FUNCTION_BLOCK T_StringSplitterEx
VAR
	SubjectString : TC2_SYSTEM.T_MaxString;
	Delimiter : STRING;
	Delimiter1 : STRING;
	Delimiter2 : STRING;
	NextDelimiterPosition : INT;
	NextDelimiter1Position : INT;
	NextDelimiter2Position : INT;
END_VAR

METHOD GetNext : STRING(255)
VAR_INPUT
END_VAR
VAR
	RemainingLength: INT;
END_VAR
NextDelimiter1Position := FIND(SubjectString , Delimiter1);
NextDelimiter2Position := FIND(SubjectString , Delimiter2);

IF NextDelimiter1Position = 0 THEN
    // use Delimiter 2 position , even if zero...
    NextDelimiterPosition := NextDelimiter2Position;
    Delimiter := Delimiter2;
    
ELSIF NextDelimiter2Position = 0 THEN
    // use Delimiter 1 position , non-zero...
    NextDelimiterPosition := NextDelimiter1Position;
    Delimiter := Delimiter1;

ELSE
    // Both delimters found - use the one nearest the start of the string...
    IF NextDelimiter1Position < NextDelimiter2Position THEN
        NextDelimiterPosition := NextDelimiter1Position;
        Delimiter := Delimiter1;
    ELSE
        NextDelimiterPosition := NextDelimiter2Position;
        Delimiter := Delimiter2;
	END_IF
END_IF

IF NextDelimiterPosition > 0 THEN // delimitter found
    
    // extract next sub-string
	GetNext := LEFT(SubjectString,NextDelimiterPosition - 1);
    
    // remove sub-string from subject string
	RemainingLength := LEN(SubjectString) - NextDelimiterPosition - LEN(Delimiter) + 1;
	SubjectString := RIGHT(SubjectString,RemainingLength);
    
    // strip any delimitters from front of remaining string
    WHILE FIND(SubjectString,Delimiter1) = 1 DO
        SubjectString := RIGHT(SubjectString,LEN(SubjectString) - LEN(Delimiter1));
	END_WHILE
    WHILE FIND(SubjectString,Delimiter2) = 1 DO
        SubjectString := RIGHT(SubjectString,LEN(SubjectString) - LEN(Delimiter2));
	END_WHILE
	
ELSE
	GetNext := SubjectString; // return what is left
	SubjectString := '';
END_IF
END_METHOD

METHOD GetRemainder : STRING(255)
GetRemainder := SubjectString; // return what is left
SubjectString := '';
END_METHOD

METHOD HasMore : BOOL
VAR_INPUT
END_VAR
HasMore := SubjectString <> '';
END_METHOD

METHOD Init
VAR_INPUT
		Str : TC2_SYSTEM.T_MaxString;
		Delim1 : STRING;
		Delim2 : STRING;
END_VAR
SubjectString := Str;
NextDelimiterPosition := 0;
Delimiter1 := Delim1;
Delimiter2 := Delim2;
END_METHOD

END_FUNCTION_BLOCK

(* stored: Version 1.1.0.1, ProductVersion 3.1.4024.15
   POU T_StringSplitterEx: Id {5351917b-6c6b-081b-3f6c-a0d5576dc9e3}, SpecialFunc None
   Method GetNext: Id {c3970227-379a-0eb8-341d-b18e20b3ac81}
   Method GetRemainder: Id {94e2acbc-ea2f-08f7-3282-27b8ef7bcce3}
   Method HasMore: Id {55004a7b-63c4-0a5a-3bb7-6f979886cd65}
   Method Init: Id {eaec9f99-fd6f-0a88-3512-94964355b0d9} *)
